ORGANIZATION_BLOCK "OB_MOD_ERR"
TITLE =
//$Revision: 1.3 $
//$Date: 2008/06/06 08:32:35CEST $
//$Author: hgc $
//
//
//"Module Access Error"

VERSION : 0.1


VAR_TEMP
  OB122_EV_CLASS : BYTE ;	//16#29, Event class 2, Entering event state, Internal fault event
  OB122_SW_FLT : BYTE ;	//16#XX Software error code
  OB122_PRIORITY : BYTE ;	//X = Priority of OB where fault occured (Priority of 1 is lowest)
  OB122_OB_NUMBR : BYTE ;	//122 (Organization block 122, OB122)
  OB122_BLK_TYPE : BYTE ;	//16#88/8A/8C/8E Type of block fault occured in
  OB122_MEM_AREA : BYTE ;	//Memory area where access error occured
  OB122_MEM_ADDR : WORD ;	//Memory address where access error occured
  OB122_BLK_NUM : WORD ;	//Block number in which error occured
  OB122_PRG_ADDR : WORD ;	//Program address where error occured
  OB122_DATE_TIME : DATE_AND_TIME ;	//Date and time OB1 started
END_VAR
BEGIN
NETWORK
TITLE =Peripheriezugriffsfehler

      U     "DB_CONFIG".ANWAHL_DURCH_USER_DATA.MASCHTYP_99_AKTIV;
      BEB   ;


      UN    "M_Ruecksetze_Fehler";
      S     "DB_FEHLERMELDUNG".Spi_VS_Halt._700312_Err_Peripherie;


      BE    ;

END_ORGANIZATION_BLOCK

